{attribute 'obsolete' := 'DUT_PositionState has been renamed to ST_PositionState'}
TYPE DUT_PositionState : ST_PositionState; END_TYPE

(* stored: Version 1.1.0.1
   DUT DUT_PositionState: Id {1162ea70-6af0-452f-8406-2ab189525e69} *)
